// TIA Portal V19 export
DATA_BLOCK "PRINT"   // DB134
{ S7_Optimized_Access := 'TRUE' }
// stored: MemoryReserve 100
   VAR RETAIN
      "PRINT START" : Bool;
   END_VAR
   VAR
      "PRESENT VALUE" : Int;
   END_VAR
   VAR RETAIN
      INTERVAL : Int;
   END_VAR
BEGIN
END_DATA_BLOCK
